                                       FOR #tempCnt := 1 TO UINT_TO_DINT(#tempRecPubTopicLength)
                                       DO
                                           IF #tempCnt < MAX_LEN(#subscriptionMessage.receivingTopic)//put everything that fits from buffer to topic output
                                           THEN
                                               #subscriptionMessage.receivingTopic[#tempCnt] := BYTE_TO_WCHAR(#statInternalBodyBuffer[#TOPIC_LEN_INFO + #tempCnt]);
                                           ELSE
                                               #subscriptionMessage.messageInvalid := TRUE;
                                               EXIT;
                                           END_IF;
                                       END_FOR;

                                       IF (#statTotalRemainingMessageLengthSaver > #MAX_INTERNAL_BUFFERLEN)//if there is a huge payload exceeding internal buffer.
                                       THEN
                                           #statTotalRemainingMessageLengthSaver := #MAX_INTERNAL_BUFFERLEN;
                                       END_IF;

                                       IF (#tempRecPubTopicLength + #TOPIC_LEN_INFO + INT_TO_UINT(#DEFAULT_TWO_BYTE_LEN) < #MAX_INTERNAL_BUFFERLEN)//len +2byte len info +2byte packetID
                                       THEN
                                           FOR #tempCnt := 1 TO UDINT_TO_DINT(#statTotalRemainingMessageLengthSaver - #TOPIC_LEN_INFO - #tempRecPubTopicLength - INT_TO_UINT(#DEFAULT_TWO_BYTE_LEN))
                                           DO
                                               IF #tempCnt < MAX_LEN(#subscriptionMessage.receivedMessageData)//put everything that fits to output message
                                               THEN
                                                   #subscriptionMessage.receivedMessageData[#tempCnt] := BYTE_TO_WCHAR(#statInternalBodyBuffer[#TOPIC_LEN_INFO + INT_TO_UINT(#DEFAULT_TWO_BYTE_LEN) + #tempRecPubTopicLength + #tempCnt]);
                                               ELSE
                                                   #subscriptionMessage.messageInvalid := TRUE;
                                                   EXIT;
                                               END_IF;
                                           END_FOR;
                                       END_IF;

                                       IF #statInternalBufferOverflow THEN
                                           #subscriptionMessage.messageInvalid := TRUE;
                                           #statInternalBufferOverflow := false;
                                       END_IF;

                                       //PUBACK - Send Publish acknowledge packet
                                       //fixed Header
                                       #statSendBufferSubscribePacketAckn[1] := INT_TO_BYTE(#MQTT_MSG_TYPE_PUBACK);
                                       #statSendBufferSubscribePacketAckn[2] := INT_TO_BYTE(#DEFAULT_TWO_BYTE_LEN);

                                       //Variable Header
                                       #statSendBufferSubscribePacketAckn[3] := #statPacketID2.%B1; //if buffer overflow, this is a guessing game
                                       #statSendBufferSubscribePacketAckn[4] := #statPacketID2.%B0;
                                       #instTcpSendSubscribedMessagesAck.LEN := INT_TO_UDINT(2 * (#DEFAULT_TWO_BYTE_LEN));

                                       #subscriptionMessage.newMessageRecieved := TRUE; //signal that new data is available
                                       #statQoS1decoded := true;
                                   ELSE
                                       //ensure its only valid for 1 cycle
                                       #subscriptionMessage.newMessageRecieved := FALSE;
                                       #subscriptionMessage.messageInvalid := FALSE;

                                   END_IF;

                                   //Verify that we are not currently sending data, else wait
                                   IF #statQoS1decoded AND NOT #instTcpSend.REQ THEN
                                       #instTcpSendSubscribedMessagesAck.REQ := true; // Start sending  data
                                   END_IF;

                                   //Wait until tsend is done
                                   IF ((#instTcpSendSubscribedMessagesAck.DONE) // wait for publish to be done.
                                       AND (#instTcpSendSubscribedMessagesAck.BUSY = false))
                                   THEN
                                       #instTcpSendSubscribedMessagesAck.REQ := false;
                                       FOR #statCnt := 1 TO (4 + 2) DO
                                           #statSendBufferSubscribePacketAckn[#statCnt] := 0; // Reset buffer
                                       END_FOR;

                                       #statStateMqttReceive := #IDLE; //reset to idle wait for new data.

                                   ELSIF #instTcpSendSubscribedMessagesAck.ERROR //If acknowledge paket failed, abort.
                                   THEN
                                       #instTcpSendSubscribedMessagesAck.REQ := false;
                                       #statStatus := #instTcpSendSubscribedMessagesAck.STATUS;
                                       #statQoS1decoded := FALSE;
                                       #statStateMqttMachine := #MQTT_ERROR_STATE;
                                       #statStatusID := #MQTT_RECEIVED_QOS1_STATE;
                                   END_IF;

                               END_REGION

                               REGION Not Yet implemented_QoS2

                                   //             #MQTT_RcvPublishQoS2:  //Receive Topic/Message QoS2 and send Publish Received / Publish complete
                                   //                 //#busy := true;
                                   //                 IF #statAlreadyExtracted = false THEN

                                   //                     #tempRecPubMsgLength := #statRcvMessageBuffer[2]; //Msg length

                                   //                     #tempRecPubTopicLength := #statRcvMessageBuffer[4]; //Topic length

                                   //                     #statPacketIDAckRecieve2.%B1 := #statRcvMessageBuffer[5 + #tempRecPubTopicLength];
                                   //                     #statPacketIDAckRecieve2.%B0 := #statRcvMessageBuffer[6 + #tempRecPubTopicLength];

                                   //                     Chars_TO_Strg(Chars := #statRcvMessageBuffer,  //extract received Msg Content 
                                   //                                   pChars := 4,
                                   //                                   Cnt := #tempRecPubTopicLength,
                                   //                                   Strg => #SubscriptionMessages.RecievedTopic);

                                   //                     Chars_TO_Strg(Chars := #statRcvMessageBuffer,  //extract received Msg Content 
                                   //                                   pChars := 6 + #tempRecPubTopicLength,
                                   //                                   Cnt := #tempRecPubMsgLength - #tempRecPubTopicLength - 4,
                                   //                                   Strg => #SubscriptionMessages.RecievedMessage);

                                   //                     #statAlreadyExtracted := True;

                                   //                     //send PUBREC publish recieved packet
                                   //                     //fixed Header
                                   //                     #statSendBufferSubscribeAckn[1] := 16#50;
                                   //                     #statSendBufferSubscribeAckn[2] := 2;
                                   //                     //Variable Header
                                   //                     #statSendBufferSubscribeAckn
                                   //                     [3] := #statPacketIDAckRecieve2.%B1;
                                   //                     #statSendBufferSubscribeAckn
                                   //                     [4] := #statPacketIDAckRecieve2.%B0;
                                   //                     #instTcpSendSubscribedMessagesAck
                                   //                     .LEN := INT_TO_UDINT(4);
                                   //                     #instTcpSendSubscribedMessagesAck
                                   //                     .REQ := true;

                                   //                 END_IF;



                                   //                 IF ((#instTcpSendSubscribedMessagesAck
                                   //                     .DONE)
                                   //                     AND (#instTcpSendSubscribedMessagesAck
                                   //                     .BUSY = false))
                                   //                 THEN
                                   //                     #instTcpSendSubscribedMessagesAck.REQ := false;
                                   //                     #statAlreadyExtracted := FALSE;
                                   //                     #statNewDataRcv := false; //signal data was already extracted.
                                   //                     #statStateMQTTReceive := #MQTT_RELAndComplete; // when paket was send, wait for response in next step

                                   //                 ELSIF #instTcpSendSubscribedMessagesAck
                                   //                     .ERROR
                                   //                 THEN
                                   //                     #statusID := #MQTT_RcvPublishQoS2;
                                   //                     #statAlreadyExtracted := FALSE;
                                   //                     #instTcpSendSubscribedMessagesAck
                                   //                     .REQ := false;
                                   //                     #statStateMQTTMachine := #MQTT_ERROR;
                                   //                     #status := #instTcpSendSubscribedMessagesAck
                                   //                     .STATUS;
                                   //                 END_IF;


                                   //             #MQTT_RELAndComplete:  //Receive Publish Release and send Publish Complete

                                   //                 IF (#statNewDataRcv AND (#statRcvMessageBuffer[1] AND 16#FF) = #MQTT_MSG_TYPE_PUBREL)
                                   //                 THEN // new data is pub release packet
                                   //                     IF //compare if packet id matches
                                   //                         (#statRcvMessageBuffer[3] = #statPacketIDAckRecieve2.%B1)
                                   //                         AND
                                   //                         (#statRcvMessageBuffer[4] = #statPacketIDAckRecieve2.%B0)
                                   //                     THEN
                                   //                         #statNewDataRcv := false;

                                   //                         //build paket PUBCOMP
                                   //                         #statSendBufferSubscribeAckn[1] := 16#70;
                                   //                         #statSendBufferSubscribeAckn[2] := 2;
                                   //                         //Variable Header
                                   //                         #statSendBufferSubscribeAckn[3] := #statPacketIDAckRecieve2.%B1;
                                   //                         #statSendBufferSubscribeAckn[4] := #statPacketIDAckRecieve2.%B0;
                                   //                         #instTcpSendSubscribedMessagesAck.LEN := INT_TO_UDINT(4);
                                   //                         #instTcpSendSubscribedMessagesAck.REQ := true;
                                   //                     ELSE
                                   //                         #statStateMQTTMachine := #MQTT_ERROR;
                                   //                         #statusID := #MQTT_RELAndComplete;
                                   //                     END_IF;
                                   //                 END_IF;

                                   //                         //wait for send publish complete 
                                   //                 IF ((#instTcpSendSubscribedMessagesAck.DONE)
                                   //                     AND (#instTcpSendSubscribedMessagesAck.BUSY = false))
                                   //                 THEN
                                   //                     // #busy := false;
                                   //                     #instTcpSendSubscribedMessagesAck.REQ := false;

                                   //                     IF NOT #statKeepAliveOff
                                   //                     THEN
                                   //                         #statTriggerKeepAlive := true;
                                   //                     END_IF;

                                   //                     #SubscriptionMessages.NewMessageArrived := TRUE;  //signal output that message arrived
                                   //                     #statStateMQTTReceive := #IDLE; // go back to idle and wait for new data;

                                   //                 ELSIF #instTcpSendSubscribedMessagesAck.ERROR
                                   //                 THEN
                                   //                     #instTcpSendSubscribedMessagesAck.REQ := false;
                                   //                     #statStateMQTTMachine := #MQTT_ERROR;
                                   //                     #status := #instTcpSendSubscribedMessagesAck.STATUS;
                                   //                 END_IF;
                               END_REGION
                       END_CASE;

                   END_REGION

                   REGION Internal Job MQTT Machine
                       // Internal MQTT Jobs: #publish / Subscribe / Unsubscribe TO Topic StateMachine
                       CASE #statStateMqttJobMachine OF
                           #IDLE:
                               REGION IDLE
                                   //Idle is only executed when TCP and MQTT are connected
                                   //and no job was orderd

                                   #statDone := false; //Clear Output and Restart PING TIMER

                                   IF #statLastState = #MQTT_ERROR_STATE
                                   THEN
                                       #statError := FALSE;
                                       //reset status and statusID aswell?
                                   END_IF;
                                   IF NOT #statEnableMqttKeepAliveTimer AND NOT #statMqttKeepAliveOff
                                   THEN
                                       #statEnableMqttKeepAliveTimer := TRUE; //start keepAliveTimer to monitor conn to server
                                   END_IF;
                               END_REGION
                           #MQTT_PUBLISH_STATE:
                               REGION JOB Publish Paket
                                   // busy already set

                                   IF LEN(IN := #publishData.publishTopic) = 0 // we cannot publish to an empty topic.
                                   THEN
                                       #statStateMqttMachine := #MQTT_ERROR_STATE;
                                       #statStatus := #MQTT_ERROR_TOPIC_EMPTY;
                                       #statStatusID := #MQTT_PUBLISH_STATE;
                                       RETURN; // skip rest as we have an error.
                                   ELSIF (#publishData.publishQoS > 2 OR #publishData.publishQoS < 0) // we can only have 0,1,2
                                   THEN
                                       #statStateMqttMachine := #MQTT_ERROR_STATE;
                                       #statStatus := #MQTT_ERROR_QOS_MISMATCH;
                                       #statStatusID := #MQTT_PUBLISH_STATE;
                                       RETURN; // skip rest as we have an error.
                                   END_IF;

                                   REGION ENCODE_DATA and start Sending

                                       IF NOT #statPubPacEncoded //set at the end, will reset when transition to next state
                                       THEN
                                           //Init Array:
                                           FILL_BLK(IN:=#EMPTY_WCHAR,
                                                    COUNT:=INT_TO_UINT(#MAX_PUBLISH_MESSAGE)+1,
                                                    OUT=>#statWStringToWCharBuffer[0]);

                                           //endInit
                                           #statConnectLengthOffset := 0;
                                           #statConnectLength := LEN(IN := #publishData.publishTopic) + LEN(IN := #publishData.publishMessageData) + #DEFAULT_TWO_BYTE_LEN;
                                           #statSendBuffer[1] := INT_TO_BYTE(#MQTT_MSG_TYPE_PUB_INC_MESSAGE_QoS0); // we modify QoS below.
                                           #statSendBuffer[1].%X0 := #publishData.publishRetainFlag;
                                           #statSendBuffer[1].%X3 := false;

                                           CASE #publishData.publishQoS OF
                                               #QOS_0:
                                                   #statSendBuffer[1].%X1 := 0;
                                                   #statSendBuffer[1].%X2 := 0;
                                               #QOS_1:
                                                   #statSendBuffer[1].%X1 := 1;
                                                   #statSendBuffer[1].%X2 := 0;
                                                   //2 Byte for Packet Identifier added
                                                   #statConnectLength := #statConnectLength + #DEFAULT_TWO_BYTE_LEN;
                                               #QOS_2:
                                                   #statSendBuffer[1].%X1 := 0;
                                                   #statSendBuffer[1].%X2 := 1;
                                                   //2 Byte for Packet Identifiert added
                                                   #statConnectLength := #statConnectLength + #DEFAULT_TWO_BYTE_LEN;
                                               ELSE:
                                                   ;
                                                   //we did catch that error above.
                                           END_CASE;

                                           #statSendLength := #statConnectLength;
                                           //determine, how much data to be send and encode as mqtt standard
                                           WHILE (#statConnectLength > 0)
                                           DO
                                               #statConnectEncodedLength := #statConnectLength MOD #CONST_128_CALC;
                                               #statConnectLength := #statConnectLength / #CONST_128_CALC;
                                               // if there are more data to encode, set the top bit of this byte
                                               IF #statConnectLength > 0
                                               THEN
                                                   //#statConnectEncodedLength := #statConnectEncodedLength OR 128;
                                                   #statConnectEncodedLength := WORD_TO_INT(INT_TO_WORD(#statConnectEncodedLength) OR INT_TO_WORD(#CONST_128_CALC));
                                                   #statSendBuffer[2 + #statConnectLengthOffset] := INT_TO_BYTE(#statConnectEncodedLength);
                                                   #statConnectLengthOffset += 1;
                                               ELSE
                                                   #statSendBuffer[2 + #statConnectLengthOffset] := INT_TO_BYTE(#statConnectEncodedLength);
                                               END_IF;
                                           END_WHILE;

                                           #statSendLength := #statSendLength + #statConnectLengthOffset;

                                           //Variable Header
                                           //Write Topic
                                           #tempLength := INT_TO_WORD(LEN(IN := #publishData.publishTopic)); //TopicLength
                                           #statSendBuffer[3 + #statConnectLengthOffset] := #tempLength.%B1;
                                           #statSendBuffer[4 + #statConnectLengthOffset] := #tempLength.%B0;

                                           Strg_TO_Chars(Strg := #publishData.publishTopic,
                                                         pChars := 0,
                                                         Cnt => #tempCountChars,
                                                         Chars := #statWStringToWCharBuffer);

                                           FOR #statCnt := 0 TO UINT_TO_INT(#tempCountChars - 1) DO
                                               #statSendBuffer[5 + #statConnectLengthOffset + #statCnt] := WCHAR_TO_BYTE(#statWStringToWCharBuffer[#statCnt]);
                                           END_FOR;
                                           #statConnectLengthOffset := #statConnectLengthOffset + DINT_TO_INT(#statCnt);

                                           //Write Data
                                           IF (#publishData.publishQoS > #QOS_0)
                                           THEN
                                               //ADD PACKET ID 
                                               #tempWordForSliceAddress := INT_TO_WORD(#statPacketID); //Packet ID as Word
                                               // Write Packet ID in to buffer
                                               #statSendBuffer[5 + #statConnectLengthOffset] := #tempWordForSliceAddress.%B1; //MSB first
                                               #statSendBuffer[6 + #statConnectLengthOffset] := #tempWordForSliceAddress.%B0; // LSB

                                               //Payload
                                               Strg_TO_Chars(Strg := #publishData.publishMessageData,
                                                             pChars := 0,
                                                             Cnt => #tempCountChars,
                                                             Chars := #statWStringToWCharBuffer);

                                               FOR #statCnt := 0 TO UINT_TO_INT(#tempCountChars - 1) DO
                                                   #statSendBuffer[7 + #statConnectLengthOffset + #statCnt] := WCHAR_TO_BYTE(#statWStringToWCharBuffer[#statCnt]);
                                               END_FOR;
                                               #instTcpSend.LEN := INT_TO_UDINT(#statSendLength + #DEFAULT_TWO_BYTE_LEN);
                                               #statPubPacEncoded := True;

                                           ELSE
                                               //NO PACKET ID
                                               Strg_TO_Chars(Strg := #publishData.publishMessageData,
                                                             pChars := 0,
                                                             Cnt => #tempCountChars,
                                                             Chars := #statWStringToWCharBuffer);

                                               FOR #statCnt := 0 TO UINT_TO_INT(#tempCountChars - 1) DO
                                                   #statSendBuffer[5 + #statConnectLengthOffset + #statCnt] := WCHAR_TO_BYTE(#statWStringToWCharBuffer[#statCnt]);
                                               END_FOR;
                                               #instTcpSend.LEN := INT_TO_UDINT(#statSendLength + #DEFAULT_TWO_BYTE_LEN);
                                               #statPubPacEncoded := true;
                                           END_IF;
                                       END_IF;

                                       //verify, that we are not currently answering a telegram.
                                       //else wait
                                       IF #statPubPacEncoded AND NOT #instTcpSendSubscribedMessagesAck.REQ
                                       THEN
                                           #instTcpSend.REQ := true; //rising edge
                                       END_IF;
                                   END_REGION

                                   // Decide next State
                                   //Started sending data, what to do:
                                   IF #instTcpSend.REQ THEN
                                       #statPubPacEncoded := False;
                                       IF (#publishData.publishQoS = #QOS_1) // check if we have more to do
                                       THEN
                                           #statPacketIDAck := #statPacketID; // we sent packetID, so copy to compare when we recieve packet
                                           #statStateMqttJobMachine := #MQTT_PUBACK_STATE;
                                       ELSIF (#publishData.publishQoS = #QOS_2)
                                       THEN
                                           #statPacketIDAck := #statPacketID; // we sent packetID, so copy to compare when we recieve packet
                                           #statStateMqttJobMachine := #MQTT_PUBREC_ACK_STATE;
                                       ELSE
                                           //QoS = 0; just wait for tsend to finish
                                           #statStateMqttJobMachine := #MQTT_PUBLISH_EVAL_STATE;
                                       END_IF;
                                   END_IF;

                               END_REGION
                           #MQTT_PUBLISH_EVAL_STATE:
                               // QoS =0
                               IF ((#instTcpSend.DONE)
                                   AND (#instTcpSend.BUSY = false))
                               THEN
                                   #instTcpSend.REQ := false; //reset TSEND
                                   FOR #statCnt := 1 TO (#statSendLength + #DEFAULT_TWO_BYTE_LEN) DO //CLEAR Sendbuffer
                                       #statSendBuffer[#statCnt] := 0;
                                   END_FOR;
                                   #statDone := true;
                                   #statBusy := false;
                                   #statStateMqttJobMachine := #IDLE;
                               ELSIF #instTcpSend.ERROR // we couldnt publish data
                               THEN
                                   #statStatusID := #MQTT_PUBLISH_STATE;
                                   #instTcpSend.REQ := false;
                                   #statStateMqttMachine := #MQTT_ERROR_STATE;
                                   #statStatus := #instTcpSend.STATUS;
                               END_IF;

                           #MQTT_PUBACK_STATE:
                               REGION Wait for PUBACK Paket
                                   //We Published a Paket with Qos1
                                   //and are still busy and wait for PUBACK

                                   IF NOT #statEnableMqttAckWatchDog
                                   THEN
                                       #statEnableMqttAckWatchDog := TRUE; //Start ACK watchdog.
                                   END_IF;

                                   //Check for tsend status of publish packet
                                   IF ((#instTcpSend.DONE)
                                       AND (#instTcpSend.BUSY = false))
                                   THEN
                                       #instTcpSend.REQ := false; //reset TSEND
                                       FOR #statCnt := 1 TO (#statSendLength + #DEFAULT_TWO_BYTE_LEN) DO //CLEAR Sendbuffer
                                           #statSendBuffer[#statCnt] := 0;
                                       END_FOR;
                                   ELSIF #instTcpSend.ERROR // we couldnt publish data
                                   THEN
                                       #statStatusID := #MQTT_PUBLISH_STATE;
                                       #instTcpSend.REQ := false;
                                       #statStateMqttMachine := #MQTT_ERROR_STATE;
                                       #statStatus := #instTcpSend.STATUS;
                                   END_IF;

                                   //Check if acknowledge packet was recieved 
                                   IF #tempPubAck
                                   THEN  //We have now data in RCVMessBuffer(3Byte properly)
                                       #statEnableMqttAckWatchDog := FALSE;
                                       #instTcpSend.REQ := false; //reset tsend
                                       IF (#statTrcvHeaderBuffer[2] AND #BIT_MASK_LOWBITS) = INT_TO_BYTE(#DEFAULT_TWO_BYTE_LEN)//remainng Length must be 2;
                                       THEN //
                                           #tempWordForSliceAddress := INT_TO_WORD(#statPacketIDAck); // convert Int Packet ID to WORD
                                           IF //Compare Packet ID
                                               (#statTrcvHeaderBuffer[3] = #tempWordForSliceAddress.%B1)
                                               AND
                                               (#statTrcvHeaderBuffer[4] = #tempWordForSliceAddress.%B0)
                                           THEN // packet ID does match - all good
                                               #statDone := true;
                                               #statBusy := false;
                                               #statStateMqttJobMachine := #IDLE; // we can go back to IDLE
                                           ELSE // Packet ID does not match
                                               #statStateMqttMachine := #MQTT_ERROR_STATE;
                                               #statStatusID := #MQTT_PUBACK_STATE;
                                               //go to error state, signal error and then go back to MQTT State Connected
                                               // In error state,  MQTT JobMachine is set to back to IDLE
                                           END_IF;
                                       ELSE // We got a PUBACK paket, but remaining length was not 2 (Error)
                                           //NOT VALID
                                           //Signal error and go to error State.
                                           #statStateMqttMachine := #MQTT_ERROR_STATE;
                                           #statStatus := #statTrcvHeaderBuffer[2];
                                           #statStatusID := #MQTT_BAD_ID;
                                           // After Error state we go to #MQTT_DISCONNECTED and Close TCP
                                       END_IF;
                                       //no Data Recieved
                                   ELSIF #instMqttAcknowledgeWatchDog.Q // keepalive triggered, no reaction from server. must close network connection.
                                   THEN
                                       #statStateMqttMachine := #MQTT_ERROR_STATE;
                                       #statStatus := #MQTT_ERROR_KEEPALIVE;
                                       #statStatusID := #MQTT_TIMEOUT_ID; // we go to time out error state and then close TCP.
                                       #statEnableMqttAckWatchDog := FALSE; // we can shut down timer now.
                                   END_IF;
                               END_REGION

                           #MQTT_PUBREC_ACK_STATE:
                               REGION Wait for PUBREC Paket 
                                   //We Published a Paket with Qos2
                                   //and are still busy and wait for PUBREC
                                   IF NOT #statEnableMqttAckWatchDog
                                   THEN
                                       #statEnableMqttAckWatchDog := TRUE; //Start ACK watchdog.
                                   END_IF;

                                   //Check for tsend status of publish packet
                                   IF ((#instTcpSend.DONE)
                                       AND (#instTcpSend.BUSY = false))
                                   THEN
                                       #instTcpSend.REQ := false; //reset TSEND
                                       FOR #statCnt := 1 TO (#statSendLength + #DEFAULT_TWO_BYTE_LEN) DO //CLEAR Sendbuffer
                                           #statSendBuffer[#statCnt] := 0;
                                       END_FOR;
                                   ELSIF #instTcpSend.ERROR // we couldnt publish data
                                   THEN
                                       #statStatusID := #MQTT_PUBLISH_STATE;
                                       #instTcpSend.REQ := false;
                                       #statStateMqttMachine := #MQTT_ERROR_STATE;
                                       #statStatus := #instTcpSend.STATUS;
                                   END_IF;

                                   IF #tempPubRec
                                   THEN   //We have now data in RCVMessBuffer(3Byte properly)
                                       #statEnableMqttAckWatchDog := FALSE;
                                       #instTcpSend.REQ := false; //reset tsend
                                       IF (#statTrcvHeaderBuffer[2] AND #BIT_MASK_LOWBITS) = INT_TO_BYTE(#DEFAULT_TWO_BYTE_LEN) //remaining Length must be 2;
                                       THEN //
                                           #tempWordForSliceAddress := INT_TO_WORD(#statPacketIDAck); // convert Int Packet ID to WORD
                                           IF //Compare Packet ID
                                               (#statTrcvHeaderBuffer[3] = #tempWordForSliceAddress.%B1)
                                               AND
                                               (#statTrcvHeaderBuffer[4] = #tempWordForSliceAddress.%B0)
                                           THEN // packet ID does match
                                               //SendAnswer
                                               // Start Sending PUBREL Paket
                                               #statStateMqttJobMachine := #MQTT_PUBREC_SEND_STATE;
                                           ELSE // Packet ID does not match
                                               #statStateMqttMachine := #MQTT_ERROR_STATE;
                                               #statStatusID := #MQTT_PUBREC_ACK_STATE;
                                               //go to error state, signal error and then go back to MQTT State Connected
                                               // In error state,  MQTT JobMachine is set to back to IDLE
                                           END_IF;
                                       ELSE // We got a PUBREC paket, but remaining length was not 2 (Error)
                                           //NOT VALID
                                           //Signal error and go to error State.
                                           #statStateMqttMachine := #MQTT_ERROR_STATE;
                                           #statStatus := #statTrcvHeaderBuffer[2];
                                           #statStatusID := #MQTT_BAD_ID;
                                           // After Error state we go to #MQTT_DISCONNECTED and Close TCP
                                       END_IF;
                                       //no Data Recieved
                                   ELSIF #instMqttAcknowledgeWatchDog.Q // keepalive triggered, no reaction from server. must close network connection.
                                   THEN
                                       #statStateMqttMachine := #MQTT_ERROR_STATE;
                                       #statStatus := #MQTT_ERROR_KEEPALIVE;
                                       #statStatusID := #MQTT_TIMEOUT_ID; // we go to time out error state and then close TCP.
                                       #statEnableMqttAckWatchDog := FALSE; // we can shut down timer now.
                                   END_IF;

                               END_REGION

                           #MQTT_PUBREC_SEND_STATE:
                               REGION Send PUBRELPaket
                                   //WHEN Data was recieved and is ok:
                                   IF NOT #instTcpSendSubscribedMessagesAck.REQ // check if we currently not answer a telegramm
                                   THEN // Start Sending PUBREL Paket
                                       //fixed Header
                                       #statSendBuffer[1] := INT_TO_BYTE(#MQTT_MSG_TYPE_PUBREL); //everything else is violation.
                                       #statSendBuffer[2] := INT_TO_BYTE(#DEFAULT_TWO_BYTE_LEN); //fixed LEN
                                       //Variable Header
                                       #tempWordForSliceAddress := INT_TO_WORD(#statPacketIDAck); // convert Int Packet ID to WORD
                                       #statSendBuffer[3] := #tempWordForSliceAddress.%B1; // same ID as in recieved Paket
                                       #statSendBuffer[4] := #tempWordForSliceAddress.%B0;
                                       #instTcpSend.LEN := INT_TO_UDINT(2 * #DEFAULT_TWO_BYTE_LEN);
                                       #instTcpSend.REQ := true;
                                       #statStateMqttJobMachine := #MQTT_PUBCOMP_STATE;
                                   END_IF;

                               END_REGION

                           #MQTT_PUBCOMP_STATE:
                               REGION Wait for PUBCOMP Paket
                                   //We Published a Paket with Qos2 and Send PUBREL PAKET
                                   //and are still busy and wait for PUBCOMP.. do we need TIMEOUT?
                                   IF NOT #statEnableMqttAckWatchDog
                                   THEN
                                       #statEnableMqttAckWatchDog := TRUE; //Start ACK watchdog.
                                   END_IF;

                                   //Wait for completion
                                   IF ((#instTcpSend.DONE) // sending done
                                       AND (#instTcpSend.BUSY = false))
                                   THEN
                                       #instTcpSend.REQ := false;
                                   ELSIF #instTcpSend.ERROR
                                   THEN // we couldnt send packet
                                       #statStatusID := #MQTT_PUBLISH_STATE;
                                       #instTcpSend.REQ := false;
                                       #statStateMqttMachine := #MQTT_ERROR_STATE;
                                       #statStatus := #instTcpSend.STATUS;
                                   END_IF;

                                   IF #tempPubComp
                                   THEN  //We have now data in RCVMessBuffer(3Byte properly)
                                       #statEnableMqttAckWatchDog := FALSE; //Reset watchdog
                                       #instTcpSend.REQ := false; //reset tsend
                                       IF (#statTrcvHeaderBuffer[2] AND #BIT_MASK_LOWBITS) = INT_TO_BYTE(#DEFAULT_TWO_BYTE_LEN)  //remainng Length must be 2;
                                       THEN //Compare Packet ID
                                           #tempWordForSliceAddress := INT_TO_WORD(#statPacketIDAck); // convert Int Packet ID to WORD
                                           IF //Compare Packet ID
                                               (#statTrcvHeaderBuffer[3] = #tempWordForSliceAddress.%B1) //Still must be the same
                                               AND
                                               (#statTrcvHeaderBuffer[4] = #tempWordForSliceAddress.%B0)
                                           THEN // packet ID does match
                                               #statDone := true;
                                               #statBusy := false;
                                               #statStateMqttJobMachine := #IDLE; // we can go back to IDLE
                                           ELSE // Packet ID does not match
                                               #statStateMqttMachine := #MQTT_ERROR_STATE;
                                               #statStatusID := #MQTT_PUBCOMP_STATE;
                                               //go to error state, signal error and then go back to MQTT State Connected
                                               // In error state,  MQTT JobMachine is set to back to IDLE
                                           END_IF;
                                       ELSE // We got a PUBCOMP paket, but remaining length was not 2 (Error)
                                           //NOT VALID
                                           //Signal error and go to error State.
                                           #statStateMqttMachine := #MQTT_ERROR_STATE;
                                           #statStatus := #statTrcvHeaderBuffer[2];
                                           #statStatusID := #MQTT_BAD_ID;
                                           // After Error state we go to #MQTT_DISCONNECTED and Close TCP
                                       END_IF;
                                       //no Data Recieved
                                   ELSIF #instMqttAcknowledgeWatchDog.Q // keepalive triggered, no reaction from server. must close network connection.
                                   THEN
                                       #statStateMqttMachine := #MQTT_ERROR_STATE;
                                       #statStatus := #MQTT_ERROR_KEEPALIVE;
                                       #statStatusID := #MQTT_TIMEOUT_ID; // we go to time out error state and then close TCP.
                                       #statEnableMqttAckWatchDog := FALSE; // we can shut down timer now.
                                   END_IF;
                               END_REGION

                           #MQTT_SUBSCRIBE_STATE:
                               REGION JOB Subscribe

                                   IF NOT #statSubPacEncoded THEN
                                       //Init Array 

                                      FILL_BLK(IN:=#EMPTY_WCHAR,
                                               COUNT:=INT_TO_UINT(#MAX_PUBLISH_MESSAGE) +1,
                                               OUT=>#statWStringToWCharBuffer[0]);


                                       IF #subscribeToTopic.subscriptionQoS < #QOS_0 OR #subscribeToTopic.subscriptionQoS > #QOS_2
                                       THEN
                                           #statStateMqttMachine := #MQTT_ERROR_STATE;
                                           #statStatusID := #MQTT_SUBSCRIBE_STATE;
                                           #statStatus := #MQTT_ERROR_QOS_MISMATCH;
                                           RETURN; // error return.
                                       ELSIF LEN(IN := #subscribeToTopic.subscriptionTopic) = 0
                                       THEN //would be a protocol violation, if no topic length
                                           #statStateMqttMachine := #MQTT_ERROR_STATE;
                                           #statStatus := #MQTT_ERROR_TOPIC_EMPTY;
                                           #statStatusID := #MQTT_SUBSCRIBE_STATE;
                                           RETURN; // error return.
                                       END_IF;
                                       #statConnectLengthOffset := 0;
                                       #statSendBuffer[1] := INT_TO_BYTE(#MQTT_MSG_TYPE_SUBSCRIBE); // header for subpacket

                                       #statConnectLength := LEN(IN := #subscribeToTopic.subscriptionTopic); //for topic length
                                       #statConnectLength := #statConnectLength + #DEFAULT_TWO_BYTE_LEN;//+2 byte for topic len parameter
                                       #statConnectLength := #statConnectLength + #DEFAULT_TWO_BYTE_LEN; //add two byte for paketID
                                       #statConnectLength += 1; //add one byte for req.QOS

                                       #statSendLength := #statConnectLength;

                                       WHILE (#statConnectLength > 0)
                                       DO
                                           #statConnectEncodedLength := #statConnectLength MOD #CONST_128_CALC;
                                           #statConnectLength := #statConnectLength / #CONST_128_CALC; // when statconnectedLEngth < 128 then equals 0
                                           // if there are more data to encode, set the top bit of this byte
                                           IF #statConnectLength > 0
                                           THEN
                                               #statConnectEncodedLength := WORD_TO_INT(INT_TO_WORD(#statConnectEncodedLength) OR INT_TO_WORD(#CONST_128_CALC));
                                               #statSendBuffer[2 + #statConnectLengthOffset] := INT_TO_BYTE(#statConnectEncodedLength);
                                               #statConnectLengthOffset += 1; //Increment
                                           ELSE
                                               #statSendBuffer[2 + #statConnectLengthOffset] := INT_TO_BYTE(#statConnectEncodedLength);
                                           END_IF;
                                       END_WHILE;

                                       #statSendLength := #statSendLength + #statConnectLengthOffset; //thats how big our tsend buffer must be.
                                       //Variable Header
                                       //Add packetID
                                       #tempWordForSliceAddress := INT_TO_WORD(#statPacketID); // convert Int Packet ID to WORD
                                       #statSendBuffer[3 + #statConnectLengthOffset] := #tempWordForSliceAddress.%B1; //MSB
                                       #statSendBuffer[4 + #statConnectLengthOffset] := #tempWordForSliceAddress.%B0;//LSB

                                       //Payload
                                       #tempLength := INT_TO_WORD(LEN(IN := #subscribeToTopic.subscriptionTopic)); //set topic len
                                       #statSendBuffer[5 + #statConnectLengthOffset] := #tempLength.%B1;
                                       #statSendBuffer[6 + #statConnectLengthOffset] := #tempLength.%B0;

                                       //convert
                                       Strg_TO_Chars(Strg := #subscribeToTopic.subscriptionTopic,
                                                     pChars := 0,
                                                     Cnt => #tempCountChars,
                                                     Chars := #statWStringToWCharBuffer);
                                       //Copy to sendbuffer
                                       FOR #statCnt := 0 TO UINT_TO_DINT(#tempCountChars - 1) DO
                                           #statSendBuffer[7 + #statConnectLengthOffset + #statCnt] := WCHAR_TO_BYTE(#statWStringToWCharBuffer[#statCnt]);
                                       END_FOR;

                                       #statConnectLengthOffset := #statConnectLengthOffset + DINT_TO_INT(#statCnt);
                                       CASE #subscribeToTopic.subscriptionQoS OF //modify the last byte in the sendbuffer if we have qos !=0;
                                           #QOS_0:
                                               #statSendBuffer[7 + #statConnectLengthOffset].%X0 := FALSE;
                                               #statSendBuffer[7 + #statConnectLengthOffset].%X1 := FALSE;
                                           #QOS_1:
                                               #statSendBuffer[7 + #statConnectLengthOffset].%X0 := TRUE;
                                               #statSendBuffer[7 + #statConnectLengthOffset].%X1 := FALSE;
                                           #QOS_2:
                                               #statSendBuffer[7 + #statConnectLengthOffset].%X0 := FALSE;
                                               #statSendBuffer[7 + #statConnectLengthOffset].%X1 := TRUE;
                                           ELSE:
                                               //shouldnt occur
                                               #statStateMqttMachine := #MQTT_ERROR_STATE;
                                               #statStatusID := #MQTT_SUBSCRIBE_STATE;
                                       END_CASE;

                                       #instTcpSend.LEN := INT_TO_UDINT(#statSendLength + #DEFAULT_TWO_BYTE_LEN);
                                       #statSubPacEncoded := true;
                                   END_IF;

                                   IF #statSubPacEncoded AND NOT #instTcpSendSubscribedMessagesAck.REQ
                                   THEN
                                       #instTcpSend.REQ := true; //rising edge;
                                       // SubPaket Send, wait for SubACK
                                       #statPacketIDAck := #statPacketID;
                                       #statSubPacEncoded := false;
                                       #statStateMqttJobMachine := #MQTT_SUBACK_STATE;
                                   END_IF;

                               END_REGION

                           #MQTT_SUBACK_STATE:
                               REGION Wait for SUBACK Paket
                                   //We send a Subscribe paket
                                   //and are still busy and wait for SUBACK.. do we need TIMEOUT?
                                   IF NOT #statEnableMqttAckWatchDog
                                   THEN
                                       #statEnableMqttAckWatchDog := TRUE; //Start ACK watchdog.
                                   END_IF;

                                   IF ((#instTcpSend.DONE)
                                       AND (#instTcpSend.BUSY = false))
                                   THEN
                                       #instTcpSend.REQ := false;
                                       FOR #statCnt := 1 TO (#statSendLength + 2) DO
                                           #statSendBuffer[#statCnt] := 0;
                                       END_FOR;
                                   ELSIF #instTcpSend.ERROR
                                   THEN
                                       #statStatusID := #MQTT_SUBSCRIBE_STATE;
                                       #instTcpSend.REQ := false;
                                       #statStateMqttMachine := #MQTT_ERROR_STATE;
                                       #statStatus := #instTcpSend.STATUS;
                                   END_IF;

                                   IF #tempSubAck
                                   THEN  //We have now data in RCVMessBuffer(4Byte properly)
                                       #statEnableMqttAckWatchDog := false;
                                       #instTcpSend.REQ := false;
                                       IF (#statTrcvHeaderBuffer[2] AND #BIT_MASK_LOWBITS) = INT_TO_BYTE(#DEFAULT_THREE_BYTE_LEN) //remainng Length must be 3;
                                       THEN //
                                           #tempWordForSliceAddress := INT_TO_WORD(#statPacketIDAck); // convert Int Packet ID to WORD
                                           IF //Compare Packet ID
                                               (#statTrcvHeaderBuffer[3] = #tempWordForSliceAddress.%B1)
                                               AND
                                               (#statTrcvHeaderBuffer[4] = #tempWordForSliceAddress.%B0)
                                           THEN // packet ID does match, check resultcode
                                               IF ((#statTrcvHeaderBuffer[5] AND #BIT_MASK_ALL) = INT_TO_BYTE(#subscribeToTopic.subscriptionQoS))
                                               THEN // requested QoS matches granted QoS
                                                   #statDone := true;
                                                   #statBusy := false;
                                                   #statStateMqttJobMachine := #IDLE; // we can go back to IDLE
                                               ELSE
                                                   #statStateMqttMachine := #MQTT_ERROR_STATE;
                                                   #statStatusID := #MQTT_SUBSCRIBE_STATE;
                                                   #statStatus := #MQTT_ERROR_SUBSCRIPTION_FAILURE;
                                               END_IF;
                                           ELSE // Packet ID does not match
                                               #statStateMqttMachine := #MQTT_ERROR_STATE;
                                               #statStatusID := #MQTT_SUBACK_STATE;
                                               //go to error state, signal error and then go back to MQTT State Connected
                                               // In error state,  MQTT JobMachine is set to back to IDLE
                                           END_IF;
                                       ELSE // We got a SUBACK paket, but remaining length was not 3 (Error)
                                           //NOT VALID
                                           //Signal error and go to error State.
                                           #statStateMqttMachine := #MQTT_ERROR_STATE;
                                           #statStatus := #statTrcvHeaderBuffer[2];
                                           #statStatusID := #MQTT_BAD_ID;
                                           // After Error state we go to #MQTT_DISCONNECTED and Close TCP
                                       END_IF;
                                       //no Data Recieved
                                   ELSIF #instMqttAcknowledgeWatchDog.Q // keepalive triggered, no reaction from server. must close network connection.
                                   THEN
                                       #statStateMqttMachine := #MQTT_ERROR_STATE;
                                       #statStatus := #MQTT_ERROR_KEEPALIVE;
                                       #statStatusID := #MQTT_TIMEOUT_ID; // we go to time out error state and then close TCP.
                                       #statEnableMqttAckWatchDog := FALSE; // we can shut down timer now.
                                   END_IF;
                               END_REGION

                           #MQTT_UNSUBSCRIBE_STATE:
                               REGION JOB Unsubscribe

                                   IF NOT #statUnsubPacEncoded THEN
                                       FILL_BLK(IN:=#EMPTY_WCHAR,
                                                COUNT:=INT_TO_UINT(#MAX_PUBLISH_MESSAGE)+1,
                                                OUT=>#statWStringToWCharBuffer[0]);


                                       IF LEN(IN := #subscribeToTopic.subscriptionTopic) = 0
                                       THEN //would be a protocol violation, if no topic length set
                                           #statStateMqttMachine := #MQTT_ERROR_STATE;
                                           #statStatusID := #MQTT_UNSUBSCRIBE_STATE;
                                           RETURN; // error return.
                                       END_IF;
                                       #statConnectLengthOffset := 0;
                                       //fixed header
                                       #statSendBuffer[1] := INT_TO_BYTE(#MQTT_MSG_TYPE_UNSUBSCRIBE); //MSG_TYPE_Unsubscribe

                                       #statConnectLength := LEN(IN := #subscribeToTopic.subscriptionTopic); //is topic length
                                       #statConnectLength := #statConnectLength + #DEFAULT_TWO_BYTE_LEN;//+2 byte for topic len parameter
                                       #statConnectLength := #statConnectLength + #DEFAULT_TWO_BYTE_LEN; //+2  byte for paketID 

                                       #statSendLength := #statConnectLength; //remaining length,before encoding. 

                                       WHILE (#statConnectLength > 0)
                                       DO
                                           #statConnectEncodedLength := #statConnectLength MOD #CONST_128_CALC;
                                           #statConnectLength := #statConnectLength / #CONST_128_CALC; // when statconnectedLEngth < 128 then equals 0
                                           // if there are more data to encode, set the top bit of this byte
                                           IF #statConnectLength > 0
                                           THEN
                                               #statConnectEncodedLength := WORD_TO_INT(INT_TO_WORD(#statConnectEncodedLength) OR INT_TO_WORD(#CONST_128_CALC));
                                               #statSendBuffer[2 + #statConnectLengthOffset] := INT_TO_BYTE(#statConnectEncodedLength);
                                               #statConnectLengthOffset := #statConnectLengthOffset + 1;
                                           ELSE
                                               #statSendBuffer[2 + #statConnectLengthOffset] := INT_TO_BYTE(#statConnectEncodedLength);
                                           END_IF;
                                       END_WHILE;

                                       #statSendLength := #statSendLength + #statConnectLengthOffset; //thats how big our tsend buffer must be.

                                       //Variable Header
                                       //Add packetID
                                       #tempWordForSliceAddress := INT_TO_WORD(#statPacketID); // convert Int Packet ID to WORD
                                       #statSendBuffer[3 + #statConnectLengthOffset] := #tempWordForSliceAddress.%B1;
                                       #statSendBuffer[4 + #statConnectLengthOffset] := #tempWordForSliceAddress.%B0;

                                       //Payload
                                       #tempLength := INT_TO_WORD(LEN(IN := #subscribeToTopic.subscriptionTopic)); //set topic len
                                       #statSendBuffer[5 + #statConnectLengthOffset] := #tempLength.%B1;
                                       #statSendBuffer[6 + #statConnectLengthOffset] := #tempLength.%B0;

                                       //convert
                                       Strg_TO_Chars(Strg := #subscribeToTopic.subscriptionTopic,
                                                     pChars := 0,
                                                     Cnt => #tempCountChars,
                                                     Chars := #statWStringToWCharBuffer);

                                       //Copy to sendbuffer
                                       FOR #statCnt := 0 TO UINT_TO_INT(#tempCountChars - 1) DO
                                           #statSendBuffer[7 + #statConnectLengthOffset + #statCnt] := WCHAR_TO_BYTE
                                           (#statWStringToWCharBuffer[#statCnt]);
                                       END_FOR;

                                       #instTcpSend.LEN := INT_TO_UDINT(#statSendLength + #DEFAULT_TWO_BYTE_LEN);
                                       #statUnsubPacEncoded := TRUE;
                                   END_IF;

                                   IF #statUnsubPacEncoded AND NOT #instTcpSendSubscribedMessagesAck.REQ // check if not answering telegram.
                                   THEN
                                       #instTcpSend.REQ := true; //rising edge;
                                       // UnSubPaket Send, wait for UnSubACK
                                       #statPacketIDAck := #statPacketID;
                                       #statUnsubPacEncoded := false;
                                       #statStateMqttJobMachine := #MQTT_UNSUBACK_STATE;
                                   END_IF;


                               END_REGION
                           #MQTT_UNSUBACK_STATE:
                               REGION Wait for UNSUBACK Packet                                     
                                   //We send a Subscribe paket
                                   //and are still busy and wait for SUBACK.. do we need TIMEOUT?
                                   IF NOT #statEnableMqttAckWatchDog
                                   THEN
                                       #statEnableMqttAckWatchDog := TRUE; //Start ACK watchdog.
                                   END_IF;

                                   //Check TSend Status
                                   IF ((#instTcpSend.DONE)
                                       AND (#instTcpSend.BUSY = false))
                                   THEN
                                       #instTcpSend.REQ := false;
                                       FOR #statCnt := 1 TO (#statSendLength + #DEFAULT_TWO_BYTE_LEN) DO
                                           #statSendBuffer[#statCnt] := 0;
                                       END_FOR;
                                   ELSIF #instTcpSend.ERROR
                                   THEN
                                       #statStatusID := #MQTT_UNSUBSCRIBE_STATE;
                                       #instTcpSend.REQ := false;
                                       #statStateMqttMachine := #MQTT_ERROR_STATE;
                                       #statStatus := #instTcpSend.STATUS;
                                       #statSubPacEncoded := false;
                                   END_IF;

                                   IF #tempUnSubAck
                                   THEN  //We have now data in RCVMessBuffer(3Byte properly)
                                       #statEnableMqttAckWatchDog := FALSE;
                                       #instTcpSend.REQ := false;
                                       IF #statTrcvHeaderBuffer[2] = INT_TO_BYTE(#DEFAULT_TWO_BYTE_LEN) //remainng Length must be 2;
                                       THEN //
                                           #tempWordForSliceAddress := INT_TO_WORD(#statPacketIDAck); // convert Int Packet ID to WORD
                                           IF //Compare Packet ID
                                               (#statTrcvHeaderBuffer[3] = #tempWordForSliceAddress.%B1)
                                               AND
                                               (#statTrcvHeaderBuffer[4] = #tempWordForSliceAddress.%B0)
                                           THEN // packet ID does match, check resultcode
                                               #statDone := true;
                                               #statBusy := false;
                                               #statStateMqttJobMachine := #IDLE; // we can go back to IDLE
                                           ELSE // Packet ID does not match
                                               #statStateMqttMachine := #MQTT_ERROR_STATE;
                                               #statStatus := #MQTT_ERROR_PACKETID;
                                               #statStatusID := #MQTT_UNSUBACK_STATE;
                                               //go to error state, signal error and then go back to MQTT State Connected
                                               // In error state,  MQTT JobMachine is set to back to IDLE
                                           END_IF;
                                       ELSE // We got a UNSUBACK paket, but remaining length was not 2 (Error)
                                           //NOT VALID
                                           //Signal error and go to error State.
                                           #statStateMqttMachine := #MQTT_ERROR_STATE;
                                           #statStatus := #statTrcvHeaderBuffer[2];
                                           #statStatusID := #MQTT_BAD_ID;
                                           // After Error state we go to #MQTT_DISCONNECTED and Close TCP
                                       END_IF;
                                       //no Data Recieved
                                   ELSIF #instMqttAcknowledgeWatchDog.Q // keepalive triggered, no reaction from server. must close network connection.
                                   THEN
                                       #statStateMqttMachine := #MQTT_ERROR_STATE;
                                       #statStatus := #MQTT_ERROR_KEEPALIVE;
                                       #statStatusID := #MQTT_TIMEOUT_ID; // we go to time out error state and then close TCP.
                                       #statEnableMqttAckWatchDog := FALSE; // we can shut down timer now.
                                   END_IF;
                               END_REGION

                           #MQTT_PING:
                               REGION PING MQTT
                                   //Build fixed Header
                                   //Message Type
                                   IF NOT #statPingPacEncoded
                                   THEN
                                       #statSendBuffer[1] := INT_TO_BYTE(#MQTT_MSG_TYPE_PING);
                                       //Remaining Lenght (must be O)
                                       #statSendBuffer[2] := 0;
                                       #instTcpSend.LEN := INT_TO_UDINT(#DEFAULT_TWO_BYTE_LEN);
                                       #statPingPacEncoded := TRUE;
                                   END_IF;
                                   IF #statPingPacEncoded AND NOT #instTcpSendSubscribedMessagesAck.REQ
                                   THEN
                                       #instTcpSend.REQ := true;
                                       #statPingPacEncoded := FALSE;
                                       #statStateMqttJobMachine := #MQTT_PINGRESP; // go to wait for response
                                   END_IF;
                               END_REGION

                           #MQTT_PINGRESP:
                               REGION PING RESP
                                   //Wait for ackno
                                   IF NOT #statEnableMqttAckWatchDog
                                   THEN
                                       #statEnableMqttAckWatchDog := TRUE; //Start ACK watchdog.
                                   END_IF;

                                   IF ((#instTcpSend.DONE)
                                       AND (#instTcpSend.BUSY = false))
                                   THEN
                                       #instTcpSend.REQ := false; //reset edge
                                       FOR #statCnt := 0 TO 1 DO //delete send buffer
                                           #statSendBuffer[#statCnt + 1] := 0;
                                       END_FOR;
                                   ELSIF #instTcpSend.ERROR // sending failed
                                   THEN
                                       #statStatusID := #MQTT_PING;
                                       #instTcpSend.REQ := false;
                                       #statStateMqttMachine := #MQTT_ERROR_STATE;
                                       #statStatus := #instTcpSend.STATUS;
                                   END_IF;

                                   IF #tempPingResp  //Wait for TRCV to signal recieved Paket
                                   THEN // Body is empty, ok
                                       #instTcpSend.REQ := false; //reset edge
                                       #statEnableMqttAckWatchDog := false;
                                       #statBusy := false;
                                       //#statTriggerMQTTKeepAlive := true;
                                       #statStateMqttJobMachine := #IDLE; // we will start keepAlive Timer again in IDLE State.
                                       //no Data Recieved
                                   ELSIF #instMqttAcknowledgeWatchDog.Q // keepalive triggered, no reaction from server. must close network connection.
                                   THEN
                                       #statStateMqttMachine := #MQTT_ERROR_STATE;
                                       #statStatus := #MQTT_ERROR_KEEPALIVE;
                                       #statStatusID := #MQTT_TIMEOUT_ID; // we go to time out error state and then close TCP.
                                       #statEnableMqttAckWatchDog := FALSE; // we can shut down timer now.
                                   END_IF;
                               END_REGION
                       END_CASE;
                   END_REGION
               END_REGION

           #MQTT_DISCONNECT_STATE:
               REGION MQTT Disconnect
                   #statBusy := True;

                   IF NOT #instTcpSend.REQ AND NOT #instTcpSendSubscribedMessagesAck.REQ
                   THEN
                       //Build fixed Header
                       //Message Type
                       #statSendBuffer[1] := INT_TO_BYTE(#MQTT_MSG_TYPE_DISCONNECT);
                       //Remaining Length (must be O)
                       #statSendBuffer[2] := 0;

                       #instTcpSend.LEN := INT_TO_UDINT(#DEFAULT_TWO_BYTE_LEN);
                       #instTcpSend.REQ := true; //Sart Sending of DISC Packet
                   END_IF;

                   IF ((#instTcpSend.DONE)
                       AND (#instTcpSend.BUSY = false))
                   THEN
                       IF NOT #enable THEN
                           #statStateTcpMachine := #TCP_DISCONNECT;
                       END_IF;
                       #instTcpSend.REQ := false;
                       #statStateMqttMachine := #MQTT_DISCONNECTED_STATE;
                       #statStateMqttJobMachine := #IDLE;
                       #statBusy := false;
                   ELSIF #instTcpSend.ERROR
                   THEN
                       IF NOT #enable THEN
                           #statStateTcpMachine := #TCP_DISCONNECT;
                       END_IF;
                       #statStatusID := #MQTT_DISCONNECT_STATE;
                       #instTcpSend.REQ := false;
                       #statStateMqttMachine := #MQTT_ERROR_STATE;
                       #statStatus := #instTcpSend.STATUS;
                   END_IF;
               END_REGION
           #MQTT_ERROR_STATE:
               REGION MQTT Error State
                   //Errorhandling MQTT
                   #statError := true;
                   #statBusy := false;
                   #statLastState := #MQTT_ERROR_STATE;
                   #statStateMqttJobMachine := #IDLE;
                   // #statStateMQTTReceive := #IDLE;
                   #statEnableMqttKeepAliveTimer := false;
                   #statQoS1decoded := FALSE;
                   CASE #statStatusID OF
                       #MQTT_CONNECT_FLAG_CHECK_STATE:
                           #statMqttEstablished := false;
                           #statStateMqttMachine := #MQTT_DISCONNECTED_STATE;
                       #MQTT_CONNECT_STATE:
                           #statMqttEstablished := false;
                           #statStatus := #instTcpSend.STATUS;
                           #statStateMqttMachine := #MQTT_DISCONNECTED_STATE;
                       #MQTT_CONNACK_STATE:
                           #statMqttEstablished := false;
                           #statStateMqttMachine := #MQTT_DISCONNECTED_STATE;
                       #MQTT_PUBLISH_STATE:
                           #statDone := false;
                           #statStateMqttMachine := #MQTT_CONNECTED_STATE;
                           //published job failed, signal to caller and go back to idle.
                       #MQTT_PUBACK_STATE, #MQTT_PUBCOMP_STATE, #MQTT_PUBREC_ACK_STATE, #MQTT_SUBACK_STATE, #MQTT_UNSUBACK_STATE:
                           #statDone := false;
                           #statStatus := #MQTT_ERROR_PACKETID;
                           #statStateMqttMachine := #MQTT_CONNECTED_STATE;
                           //Acknowledge failed, signal to caller and go back to idle.
                       #MQTT_SUBSCRIBE_STATE, #MQTT_UNSUBSCRIBE_STATE:
                           #statDone := false;
                           #statStateMqttMachine := #MQTT_CONNECTED_STATE;
                           //Subscribe job failed, signal to caller and go back to idle.
                       #MQTT_QOS_MISMATCH_ID:
                           #statDone := false;
                           #statStatus := #MQTT_ERROR_QOS_MISMATCH;
                           #statStateMqttMachine := #MQTT_CONNECTED_STATE;
                       #MQTT_RECEIVED_QOS1_STATE:
                           #statDone := false;
                           #statStateMqttMachine := #MQTT_DISCONNECT_STATE;
                       #MQTT_PINGRESP:
                           ;
                       #MQTT_PING:
                           //we tried to send a ping paket, but tsend failed.
                           //might aswell close TCP.
                           #statMqttEstablished := false;
                           #statStatus := #instTcpSend.STATUS;
                           #statStateMqttMachine := #MQTT_DISCONNECTED_STATE;
                           #statStateTcpMachine := #TCP_DISCONNECT; //Close TCP Connection
                           ;
                       #MQTT_DISCONNECTED_STATE:
                           #statMqttEstablished := false;
                           ;
                       #MQTT_TIMEOUT_ID, #MQTT_BAD_ID:
                           #statMqttEstablished := false;
                           #statStateMqttMachine := #MQTT_DISCONNECTED_STATE;
                           #statStateTcpMachine := #TCP_DISCONNECT; //Close TCP Connection
                       ELSE
                           ;
                   END_CASE;
               END_REGION
       END_CASE;
   END_REGION


   REGION Set FB Outputs    
       // 
       //Set static variables to outputs;
       //
       #done := #statDone;
       #busy := #statBusy;
       #error := #statError;
       #status := #statStatus;
       #statusID := #statStatusID;
       #tcpEstablished := #statTcpEstablished;
       #mqttEstablished := #statMqttEstablished;

   END_REGION
END_FUNCTION_BLOCK

// ===== library types =====

// folder: Signal_Generators

FUNCTION_BLOCK "LGF_SinusCI"   // FB10027, SCL
{ S7_Optimized_Access := 'TRUE' }
VERSION : 0.1
   VAR_INPUT
      amplitude : Real := 0.0;   // Amplitude
      offset : Real := 1000.0;   // Offset
      periodeMS : UDInt := 1000;   // Periode in milliseconds
      callOB : OB_Cyclic;   // Call OB
      reset : Bool;   // Reset values
   END_VAR
   VAR_OUTPUT
      sinusValues : Real;   // Calculated Sinus values
      error : Bool;   // "0" = no error; "1" = error
      statusID : UInt;   // Error source
      status : Word;   // Status and error codes
   END_VAR
   VAR
      statRad : Real;   // Size of an angle in radians
      statCounter : UDInt;   // Counter value
   END_VAR
   VAR_TEMP
      tempCycleTime : UDInt;   // Temp cycle time from CallOB
      tempCyclePhase : UDInt;   // Temp cycle phase from CallOB
      tempCycleStatus : Word;   // Temp cycle status from CallOB
      tempReadTimeStatus : Int;   // Return value of QRY_CINT
   END_VAR
   VAR CONSTANT
      PI : Real := 3.141593;   // PI
      NO_ERROR : Word := 16#0000;   // Status no error
      OB_UNAVAILABLE : Word := 16#8200;   // Status OB not available
      ERROR_IN_THIS_BLOCK : UInt := 1;   // Error ID local error
      ERROR_QRY_CINT : UInt := 2;   // Error ID error in function QRY_CINT
   END_VAR
BEGIN
   //=============================================================================
   // Siemens AG
   // (c)Copyright 2017
   //-----------------------------------------------------------------------------
   // Library:       LGF (Library General Functions)
   // Tested with:   CPU1212C DC/DC/DC FW:V4.2
   // Engineering:   TIA Portal V15 Upd 2
   // Restrictions:  -
   // Requirements:  PLC (S7-1200 / S7-1500)
   // Functionality: This function generates a sinus signal
   //-----------------------------------------------------------------------------
   // Change log table:
   // Version  Date        In charge/Changes applied
   // 01.00.00 03.07.2018  Siemens Industry Online Support
   //                      First released version
   // 01.00.01 17.08.2018  Siemens Industry Online Support
   //                      Upgrade: TIA V15 Update 2
   //-----------------------------------------------------------------------------
   //Status Codes: -
   //=============================================================================

   // Initialize
   #error := FALSE;
   #statusID := #ERROR_IN_THIS_BLOCK;
   #status := #NO_ERROR;

   // get sample time, according to the cyclic interrupt OB number
   #tempReadTimeStatus := QRY_CINT(OB_NR := #callOB, CYCLE => #tempCycleTime,
                                   PHASE => #tempCyclePhase, STATUS => #tempCycleStatus);

   // Generate error message of the QRY_CINT function
   IF (#tempReadTimeStatus <> 0)
   THEN
     #error := TRUE;
     #statusID := #ERROR_QRY_CINT;
     #status := INT_TO_WORD(#tempReadTimeStatus);
     RETURN;
   END_IF;

   // Generate error message when OB unavailable
   IF (#tempCycleStatus = 16#0000)
   THEN
     #error := TRUE;
     #statusID := #ERROR_IN_THIS_BLOCK;
     #status := #OB_UNAVAILABLE;
     RETURN;
   END_IF;

   IF (#reset = TRUE)
   THEN
     #statCounter := 0;
     #sinusValues := 0;
   ELSE
     // Increment Counter with each call of "OB_Cyclic_interrupt"
     #statCounter := #statCounter + (#tempCycleTime) / 1000;
     #statCounter := #statCounter MOD (#periodeMS);

     #statRad := UDINT_TO_REAL(#statCounter) * 2.0 * #PI / (UDINT_TO_REAL(#periodeMS));

     #sinusValues := SIN(#statRad) * #amplitude + #offset;
   END_IF;
END_FUNCTION_BLOCK

FUNCTION_BLOCK "LGF_RectangleCI"   // FB10029, SCL
{ S7_Optimized_Access := 'TRUE' }
VERSION : 0.1
   VAR_INPUT
      amplitude : Real := 0.0;   // Amplitude
      offset : Real := 1000.0;   // Offset
      periodeMS : UDInt := 1000;   // Periode in milliseconds
      callOB : OB_Cyclic;   // Call OB
      reset : Bool;   // Reset values
   END_VAR
   VAR_OUTPUT
      rectangleValues : Real;   // Calculated rectangle values
      error : Bool;   // "0" = no error; "1" = error
      statusID : UInt;   // Error source
      status : Word;   // Status and error codes
   END_VAR
   VAR
      statRad : Real;   // Size of an angle in radians
      statCounter : UDInt;   // Counter value
   END_VAR
   VAR_TEMP
      tempCycleTime : UDInt;   // Temp cycle time from CallOB
      tempCyclePhase : UDInt;   // Temp cycle phase from CallOB
      tempCycleStatus : Word;   // Temp cycle status from CallOB
      tempReadTimeStatus : Int;   // Return value of QRY_CINT
   END_VAR
   VAR CONSTANT
      PI : Real := 3.141593;   // PI
      NO_ERROR : Word := 16#0000;   // Status no error
      OB_UNAVAILABLE : Word := 16#8200;   // Status OB not available
      ERROR_IN_THIS_BLOCK : UInt := 1;   // Error ID local error
      ERROR_QRY_CINT : UInt := 2;   // Error ID error in function QRY_CINT
   END_VAR
BEGIN
   //=============================================================================
   // Siemens AG
   // (c)Copyright 2017
   //-----------------------------------------------------------------------------
   // Library:       LGF (Library General Functions)
   // Tested with:   CPU1212C DC/DC/DC FW:V4.2
   // Engineering:   TIA Portal V15 Upd 2
   // Restrictions:  -
   // Requirements:  PLC (S7-1200 / S7-1500)
   // Functionality: This function generates a rectangle signal
   //-----------------------------------------------------------------------------
   // Change log table:
   // Version  Date        In charge/Changes applied
   // 01.00.00 03.07.2018  Siemens Industry Online Support
   //                      First released version
   // 01.00.01 17.08.2018  Siemens Industry Online Support
   //                      Upgrade: TIA V15 Update 2
   //-----------------------------------------------------------------------------
   //Status Codes: -
   //=============================================================================

   // Initialize
   #error := FALSE;
   #statusID := #ERROR_IN_THIS_BLOCK;
   #status := #NO_ERROR;

   // get sample time, according to the cyclic interrupt OB number
   #tempReadTimeStatus := QRY_CINT(OB_NR := #callOB, CYCLE => #tempCycleTime,
                                   PHASE => #tempCyclePhase, STATUS => #tempCycleStatus);

   // Generate error message of the QRY_CINT function
   IF (#tempReadTimeStatus <> 0)
   THEN
     #error := TRUE;
     #statusID := #ERROR_QRY_CINT;
     #status := INT_TO_WORD(#tempReadTimeStatus);
     RETURN;
   END_IF;

   // Generate error message when OB unavailable
   IF (#tempCycleStatus = 16#0000)
   THEN
     #error := TRUE;
     #statusID := #ERROR_IN_THIS_BLOCK;
     #status := #OB_UNAVAILABLE;
     RETURN;
   END_IF;

   IF (#reset = TRUE) 
   THEN
     #statCounter := 0;
     #rectangleValues := 0;
   ELSE
     // Increment Counter with each call of "OB_Cyclic_interrupt"
     #statCounter := #statCounter + (#tempCycleTime) / 1000;
     #statCounter := #statCounter MOD (#periodeMS);

     IF (#statCounter <= (#periodeMS / 2))
     THEN
       #rectangleValues := #offset + #amplitude;
     ELSE
       #rectangleValues := #offset - #amplitude;
     END_IF;
   END_IF;
END_FUNCTION_BLOCK

FUNCTION "LGF_RandomInt" : Int   // FC10013, SCL
{ S7_Optimized_Access := 'TRUE' }
   VAR_INPUT
      minValue : Int;   // minimal Value random can reach
      maxValue : Int;   // maximal Value random can reach
   END_VAR
   VAR_OUTPUT
      error : Bool;
      statusID : UInt;
      status : Word;
   END_VAR
   VAR_TEMP
      tempTime : DTL;
      tempTimeStatus : Int;
      tempRandomValue : Int;
      tempNormReal : Real;
   END_VAR
   VAR CONSTANT
      NO_ERROR : Word := 16#0000;
      NO_CURRENT_JOBS : Word := 16#7000;
      MAX_LESS_MIN : Word := 16#8200;
      ERROR_IN_THIS_BLOCK : UInt := 1;
      ERROR_RD_SYS_T : UInt := 2;
      MIN_INT : DInt := -32768;
      MAX_INT : DInt := 32767;
   END_VAR
BEGIN
   //=============================================================================
   // Siemens AG
   // (c)Copyright 2017
   //-----------------------------------------------------------------------------
   // Library:       LGF (Library General Functions)
   // Tested with:   CPU1212C DC/DC/DC FW:V4.2
   // Engineering:   TIA Portal V13 SP1 Upd 4
   // Restrictions:  -
   // Requirements:  PLC (S7-1200 / S7-1500)
   // Functionality: This function generates random numbers in defined limits
   //                (Datatype Int)
   //-----------------------------------------------------------------------------
   // Change log table:
   // Version  Date        In charge / Changes applied
   // 01.00.00 19.08.2015  Siemens Industry Online Support
   //                      First released version
   // 01.00.01 02.01.2017  Siemens Industry Online Support
   //                      Upgrade: TIA Portal V14 Update 1
   // 01.00.02 17.08.2018  Siemens Industry Online Support
   //                      Upgrade: TIA V15 Update 2
   //-----------------------------------------------------------------------------
   //Status Codes:
   // 16#7000:  No current jobs
   // 16#0000:  Job finished; Note: There is no "Busy"-Status because the block
   //           is finished within a single cycle
   // 16#8200:  maxValue is samller then minValue 
   //=============================================================================

   //Set "No current job" status
   #error := false;
   #statusID := #ERROR_IN_THIS_BLOCK;
   #status := #NO_CURRENT_JOBS;

   //Check if the maximal Value is less than the minimal value
   IF (#minValue > #maxValue) THEN
     #error := true;
     #statusID := #ERROR_IN_THIS_BLOCK;
     #status := #MAX_LESS_MIN;
     #LGF_RandomInt := 0;
     RETURN;
   END_IF;

   //Read system time
   #tempTimeStatus := RD_SYS_T(#tempTime);

   IF (#tempTimeStatus <> 0) THEN
     #error := true;
     #statusID := #ERROR_RD_SYS_T;
     #status := INT_TO_WORD(#tempTimeStatus);
     #LGF_RandomInt := 0;
     RETURN;
   END_IF;

   //Callculate a random-start-value depending on the time
   #tempRandomValue.%B1 := #tempTime.NANOSECOND.%B0;
   #tempRandomValue.%B0 := #tempTime.NANOSECOND.%B1;

   //adapt the calculated random number to the given number span
   #tempNormReal := NORM_X(MIN := #MIN_INT, VALUE := #tempRandomValue, MAX := #MAX_INT);
   #LGF_RandomInt := SCALE_X(MIN := #minValue, VALUE := #tempNormReal, MAX := #maxValue);

   #status := #NO_ERROR;
END_FUNCTION